KUKA KRL program: chk_w5_grp1_clo.src, chk_w5_grp1_clo.dat

--- chk_w5_grp1_clo.src ---
&ACCESS RV4
&REL 15
&COMMENT Check grp Z1 fechado AXOR
&PARAM TEMPLATE = C:\KRC\Roboter\Template\vorgabe
&PARAM EDITMASK = *
DEF chk_w5_grp1_clo( )
;FOLD ; Programa de verificacao de grampos Z1 fechado AXOR;%{PE}%R 4.1.16,%MKUKATPBASIS,%CCOMMENT,%VNORMAL,%P 2:Programa de verificacao de grampos Z1 fechado AXOR
;ENDFOLD

$TIMER[10] = 0
$TIMER_STOP[10] = FALSE

;FOLD WAIT FOR ( NOT IN 499 'Z1.1 ABERTO' );%{PE}%R 8.2.24,%MKUKATPBASIS,%CEXT_WAIT_FOR,%VEXT_WAIT_FOR,%P 2:, 4:NOT, 5:$IN, 6:499, 7:Z1.1 ABERTO, 9:
WAIT FOR  (  NOT $IN[499] )
;ENDFOLD
;FOLD WAIT FOR ( NOT IN 501 'Z1.2 ABERTO' );%{PE}%R 8.2.24,%MKUKATPBASIS,%CEXT_WAIT_FOR,%VEXT_WAIT_FOR,%P 2:, 4:NOT, 5:$IN, 6:501, 7:Z1.2 ABERTO, 9:
WAIT FOR  (  NOT $IN[501] )
;ENDFOLD
;FOLD WAIT FOR ( NOT IN 503 'Z1.3 ABERTO' );%{PE}%R 8.2.24,%MKUKATPBASIS,%CEXT_WAIT_FOR,%VEXT_WAIT_FOR,%P 2:, 4:NOT, 5:$IN, 6:503, 7:Z1.3 ABERTO, 9:
WAIT FOR  (  NOT $IN[503] )
;ENDFOLD
;FOLD WAIT FOR ( IN 500 'Z1.1 FECHADO' );%{PE}%R 8.2.24,%MKUKATPBASIS,%CEXT_WAIT_FOR,%VEXT_WAIT_FOR,%P 2:, 4:, 5:$IN, 6:500, 7:Z1.1 FECHADO, 9:
WAIT FOR  ( $IN[500] )
;ENDFOLD
;FOLD WAIT FOR ( IN 502 'Z1.2 FECHADO' );%{PE}%R 8.2.24,%MKUKATPBASIS,%CEXT_WAIT_FOR,%VEXT_WAIT_FOR,%P 2:, 4:, 5:$IN, 6:502, 7:Z1.2 FECHADO, 9:
WAIT FOR  ( $IN[502] )
;ENDFOLD
;FOLD WAIT FOR ( IN 504 'Z1.3 FECHADO' );%{PE}%R 8.2.24,%MKUKATPBASIS,%CEXT_WAIT_FOR,%VEXT_WAIT_FOR,%P 2:, 4:, 5:$IN, 6:504, 7:Z1.3 FECHADO, 9:
WAIT FOR  ( $IN[504] )
;ENDFOLD

$TIMER_STOP[10] = TRUE
$TIMER[10] = 0

END

--- chk_w5_grp1_clo.dat ---
&ACCESS RV4
&REL 15
&COMMENT Check grp Z1 fechado AXOR
&PARAM TEMPLATE = C:\KRC\Roboter\Template\vorgabe
&PARAM EDITMASK = *
DEFDAT  CHK_W5_GRP1_CLO
;FOLD EXTERNAL DECLARATIONS;%{PE}%V3.2.0,%MKUKATPBASIS,%CEXT,%VCOMMON,%P
;FOLD BAS EXT;%{PE}%V3.2.0,%MKUKATPBASIS,%CEXT,%VEXT,%P
EXT  BAS (BAS_COMMAND  :IN,REAL  :IN )
DECL INT SUCCESS
;ENDFOLD
;FOLD GRIPPER EXT;%{E}%V3.2.0,%MKUKATPGRIPPER,%CEXT,%VEXT,%P
EXT  H50 (INT  :IN,INT  :IN,INT  :IN,GRP_TYP  :IN )
;ENDFOLD
;FOLD SPOT EXT;%{E}%V3.2.0,%MKUKATPSPOT,%CEXT,%VEXT,%P
EXT  USERSPOT (S_COMMAND  :IN,SPOT_TYPE  :IN )
;ENDFOLD
;FOLD USER EXT;%{E}%V3.2.0,%MKUKATPUSER,%CEXT,%VEXT,%P
;Make here your modifications
;ENDFOLD
;ENDFOLD

DECL BASIS_SUGG_T LAST_BASIS={POINT1[] "P0                      ",POINT2[] "P0                      ",CP_PARAMS[] "CPDAT0                  ",PTP_PARAMS[] "PDAT0                   ",CONT[] "                        ",CP_VEL[] "2.0                     ",PTP_VEL[] " 100                    "}
ENDDAT
